// TIA Portal V19 export
FUNCTION_BLOCK "Projekt_2B_Robotgrinder"   // FB4, LAD
{ S7_Optimized_Access := 'TRUE' }
// stored: MemoryReserve 100, SetENOAutomatically false
   VAR_INPUT
      Emergency_Stop_Status_150K1 : Bool;
      Sensor_102B2 : Bool;
      Sensor_102B3 : Bool;
      Sensor_102B4 : Bool;
      Sensor_102B5 : Bool;
      Sensor_102B6 : Bool;
      HMI_Start : Bool;
      HMI_Pause : Bool;
      HMI_Reset : Bool;
      HMI_Start_1 : Bool;
      HMI_Pause_1 : Bool;
      HMI_Reset_1 : Bool;
      Pause_Process : Bool;
   END_VAR
   VAR_OUTPUT
      Valve_106Q6 : Bool;
      Motor_4Q3 : Bool;
      Motor_4Q5 : Bool;
      Motor_6Q1 : Bool;
      Motor_6Q3 : Bool;
      Reset_Safety_150K1 : Bool;
   END_VAR
   VAR
      Main_Step : Int;
      Process_Step : Int;
      Reset_Step : Int;
      Placement_Step : Int;
      Order_Amount : Int;
      Items_Produced : Int;
      Items_Delivered : Int;
      Total_orders : Int;
      Storage_Amount : Int;
      Storage_Plus_Produce : Int;
      Storage_Min : Int;
      Storage_Max : Int;
      Robot_Done : Bool;
   END_VAR
BEGIN

REGION Network 1: Main Process Step 0
   // If the system is currently idling, then pressing start will start the process. On PLC restart, moves starting values into steps.
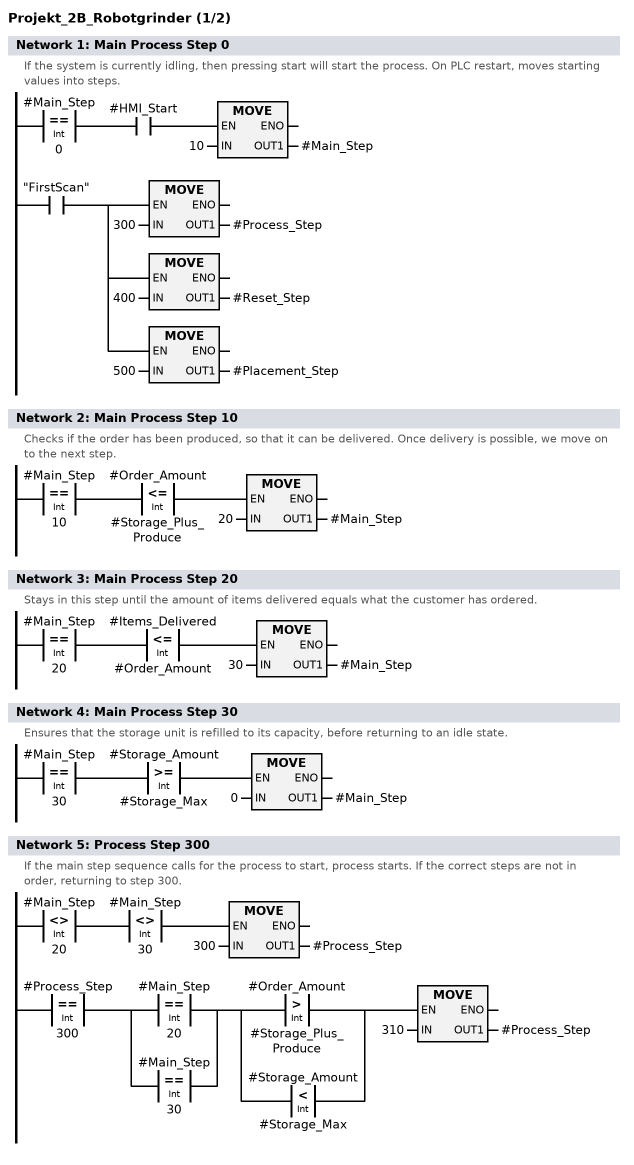
   RUNG wire#powerrail
      { S7_Templates := "SrcType := Int" } EQ_Contact(in1 := #Main_Step, in2 := 0)
      Contact( #HMI_Start )
      Move(in := 10, out1 => #Main_Step)
   END_RUNG
   RUNG wire#powerrail
      Contact( "FirstScan" )
      wire#w1
      Move(in := 300, out1 => #Process_Step)
   END_RUNG
   RUNG wire#w1
      Move(in := 400, out1 => #Reset_Step)
   END_RUNG
   RUNG wire#w1
      Move(in := 500, out1 => #Placement_Step)
   END_RUNG
   // the same network as SCL:
   IF (#Main_Step = 0) AND #HMI_Start THEN #Main_Step := 10; END_IF;
   IF "FirstScan" THEN
       #Process_Step := 300;
       #Reset_Step := 400;
       #Placement_Step := 500;
   END_IF;
END_REGION

REGION Network 2: Main Process Step 10
   // Checks if the order has been produced, so that it can be delivered. Once delivery is possible, we move on to the next step.
   RUNG wire#powerrail
      { S7_Templates := "SrcType := Int" } EQ_Contact(in1 := #Main_Step, in2 := 10)
      { S7_Templates := "SrcType := Int" } LE_Contact(in1 := #Order_Amount, in2 := #Storage_Plus_Produce)
      Move(in := 20, out1 => #Main_Step)
   END_RUNG
   // the same network as SCL:
   IF (#Main_Step = 10) AND (#Order_Amount <= #Storage_Plus_Produce) THEN #Main_Step := 20; END_IF;
END_REGION

REGION Network 3: Main Process Step 20
   // Stays in this step until the amount of items delivered equals what the customer has ordered.
   RUNG wire#powerrail
      { S7_Templates := "SrcType := Int" } EQ_Contact(in1 := #Main_Step, in2 := 20)
      { S7_Templates := "SrcType := Int" } LE_Contact(in1 := #Items_Delivered, in2 := #Order_Amount)
      Move(in := 30, out1 => #Main_Step)
   END_RUNG
   // the same network as SCL:
   IF (#Main_Step = 20) AND (#Items_Delivered <= #Order_Amount) THEN #Main_Step := 30; END_IF;
END_REGION

REGION Network 4: Main Process Step 30
   // Ensures that the storage unit is refilled to its capacity, before returning to an idle state.
   RUNG wire#powerrail
      { S7_Templates := "SrcType := Int" } EQ_Contact(in1 := #Main_Step, in2 := 30)
      { S7_Templates := "SrcType := Int" } GE_Contact(in1 := #Storage_Amount, in2 := #Storage_Max)
      Move(in := 0, out1 => #Main_Step)
   END_RUNG
   // the same network as SCL:
   IF (#Main_Step = 30) AND (#Storage_Amount >= #Storage_Max) THEN #Main_Step := 0; END_IF;
END_REGION

REGION Network 5: Process Step 300
   // If the main step sequence calls for the process to start, process starts. If the correct steps are not in order, returning to step 300.
   RUNG wire#powerrail
      { S7_Templates := "SrcType := Int" } NE_Contact(in1 := #Main_Step, in2 := 20)
      { S7_Templates := "SrcType := Int" } NE_Contact(in1 := #Main_Step, in2 := 30)
      Move(in := 300, out1 => #Process_Step)
   END_RUNG
   RUNG wire#powerrail
      { S7_Templates := "SrcType := Int" } EQ_Contact(in1 := #Process_Step, in2 := 300)
      wire#w1
      { S7_Templates := "SrcType := Int" } EQ_Contact(in1 := #Main_Step, in2 := 20)
      wire#w2
      { S7_Templates := "SrcType := Int" } GT_Contact(in1 := #Order_Amount, in2 := #Storage_Plus_Produce)
      wire#w3
      Move(in := 310, out1 => #Process_Step)
   END_RUNG
   RUNG wire#w1
      { S7_Templates := "SrcType := Int" } EQ_Contact(in1 := #Main_Step, in2 := 30)
   END_RUNG wire#w2
   RUNG wire#w2
      { S7_Templates := "SrcType := Int" } LT_Contact(in1 := #Storage_Amount, in2 := #Storage_Max)
   END_RUNG wire#w3
   // the same network as SCL:
   IF (#Main_Step <> 20) AND (#Main_Step <> 30) THEN #Process_Step := 300; END_IF;
   IF (#Process_Step = 300) AND ((#Main_Step = 20) OR (#Main_Step = 30)) AND ((#Order_Amount > #Storage_Plus_Produce) OR (#Storage_Amount < #Storage_Max)) THEN
       #Process_Step := 310;
   END_IF;
END_REGION

REGION Network 6: Process Step 310
   // Feeder activates in step 310. Once sensor activates by item on conveyor, moving to next step.
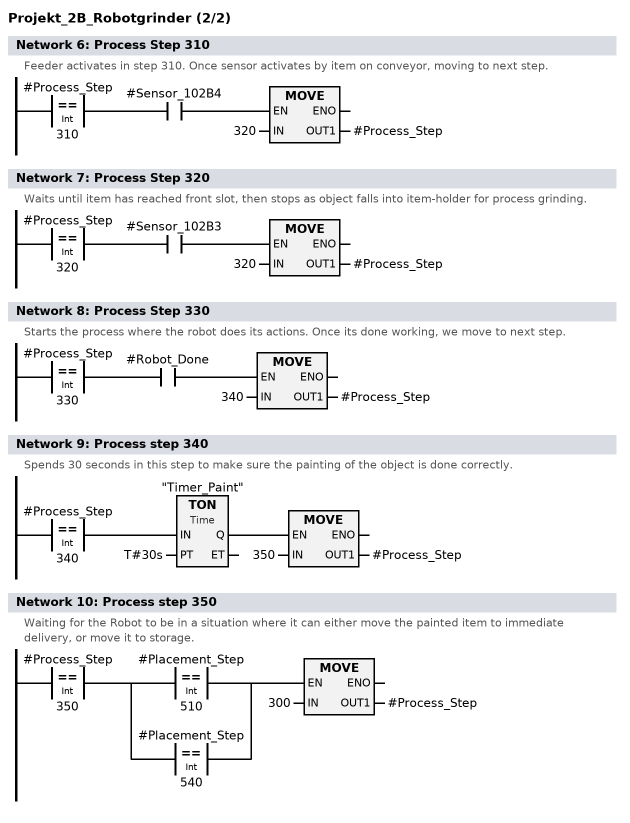
   RUNG wire#powerrail
      { S7_Templates := "SrcType := Int" } EQ_Contact(in1 := #Process_Step, in2 := 310)
      Contact( #Sensor_102B4 )
      Move(in := 320, out1 => #Process_Step)
   END_RUNG
   // the same network as SCL:
   IF (#Process_Step = 310) AND #Sensor_102B4 THEN #Process_Step := 320; END_IF;
END_REGION

REGION Network 7: Process Step 320
   // Waits until item has reached front slot, then stops as object falls into item-holder for process grinding.
   RUNG wire#powerrail
      { S7_Templates := "SrcType := Int" } EQ_Contact(in1 := #Process_Step, in2 := 320)
      Contact( #Sensor_102B3 )
      Move(in := 320, out1 => #Process_Step)
   END_RUNG
   // the same network as SCL:
   IF (#Process_Step = 320) AND #Sensor_102B3 THEN #Process_Step := 320; END_IF;
END_REGION

REGION Network 8: Process Step 330
   // Starts the process where the robot does its actions. Once its done working, we move to next step.
   RUNG wire#powerrail
      { S7_Templates := "SrcType := Int" } EQ_Contact(in1 := #Process_Step, in2 := 330)
      Contact( #Robot_Done )
      Move(in := 340, out1 => #Process_Step)
   END_RUNG
   // the same network as SCL:
   IF (#Process_Step = 330) AND #Robot_Done THEN #Process_Step := 340; END_IF;
END_REGION

REGION Network 9: Process step 340
   // Spends 30 seconds in this step to make sure the painting of the object is done correctly.
   RUNG wire#powerrail
      { S7_Templates := "SrcType := Int" } EQ_Contact(in1 := #Process_Step, in2 := 340)
      { S7_Templates := "time_type := Time" } "Timer_Paint".TON(pt := T#30s, et =>)
      Move(in := 350, out1 => #Process_Step)
   END_RUNG
   // the same network as SCL:
   "Timer_Paint".TON(IN := #Process_Step = 340, PT := T#30s);
   IF "Timer_Paint".Q THEN #Process_Step := 350; END_IF;
END_REGION

REGION Network 10: Process step 350
   // Waiting for the Robot to be in a situation where it can either move the painted item to immediate delivery, or move it to storage.
   RUNG wire#powerrail
      { S7_Templates := "SrcType := Int" } EQ_Contact(in1 := #Process_Step, in2 := 350)
      wire#w1
      { S7_Templates := "SrcType := Int" } EQ_Contact(in1 := #Placement_Step, in2 := 510)
      wire#w2
      Move(in := 300, out1 => #Process_Step)
   END_RUNG
   RUNG wire#w1
      { S7_Templates := "SrcType := Int" } EQ_Contact(in1 := #Placement_Step, in2 := 540)
   END_RUNG wire#w2
   // the same network as SCL:
   IF (#Process_Step = 350) AND ((#Placement_Step = 510) OR (#Placement_Step = 540)) THEN
       #Process_Step := 300;
   END_IF;
END_REGION
END_FUNCTION_BLOCK
